PROGRAM MAIN
VAR
END_VAR

END_PROGRAM

(* stored: Version 1.1.0.1
   POU MAIN: Id {72d29608-50da-4d49-af8d-c9a2d2e7af3b} *)
